(* PLC project CoDeSys External Library Template, WAGO e!COCKPIT e!COCKPIT, author 3S - Smart Software Solutions GmbH *)
(* stored: creationDateTime 2019-10-29T12:37:19.5035376, version 3.5.5.30, modificationDateTime 2019-10-29T12:36:39.3744516, organization 3S - Smart Software Solutions GmbH *)
(* Library project template with all possible element types, docu and a sample project structure *)

{attribute 'qualified_only'}
{attribute 'strict'}
TYPE enumSystemErrorKlasa : (BrakHeartbetuzIZE := enumKlasaAlarmu.Krytyczny, NiezgodnaIloscKomunikatowOdebranychZIZE := enumKlasaAlarmu.Systemowy, BladCRCWKomunikacieZIZE := enumKlasaAlarmu.Systemowy, BladSzyfrowania := enumKlasaAlarmu.Systemowy, ZaDuzaIloscKomunikatowWBuforze := enumKlasaAlarmu.Systemowy, BladWalidacjiFullIdentifier := enumKlasaAlarmu.Systemowy, BladFullIdentifierWHeartBeat := enumKlasaAlarmu.Systemowy, BlokadaWysylaniaRamek := enumKlasaAlarmu.Systemowy);
END_TYPE
